// TIA Portal V20 export
ORGANIZATION_BLOCK "Startup"   // OB1030, LAD, Startup
TITLE = "Complete Restart"
// stored: AutoNumber false, IsIECCheckEnabled true, Namespace Unit1.Em5, SetENOAutomatically true
   VAR_INPUT
      LostRetentive : Bool;   // True if retentive data are lost
      LostRTC : Bool;   // True if date and time are lost
   END_VAR
BEGIN

REGION Network 1 (SCL): Build the Absolut Reference Designator
   // Set the Absoult Reference Designator in the Config DB
   IF LEN(IN := "Unit1.Em5.Config".em.referenceDesignator.parent) <> 0 THEN
       "Unit1.Em5.Config".em.referenceDesignator.combined := CONCAT_WSTRING(IN1 := "Unit1.Em5.Config".em.referenceDesignator.parent, IN2 := WSTRING#'.', IN3 := "Unit1.Em5.Config".em.referenceDesignator.relative);
   ELSE
       "Unit1.Em5.Config".em.referenceDesignator.combined := "Unit1.Em5.Config".em.referenceDesignator.relative;
   END_IF;
END_REGION

REGION Network 2 (SCL): Assign axes data
   // This is an example how to assign axes to DB_ANY in DB Config. If you have axes, assign them here. The Config.axis[] variables will be handed over to the control modules. That enables a flexible programming.
   // Assign axes
   "Unit1.Em5.Config".axis[1] := "BA010AZCRDR7_NgManualInputAxisY";
   "Unit1.Em5.Config".axis[2] := "BA010AZCRDR8_MagazineAxisZ";

   // HW_SubModule
   "Unit1.Em5.Config".moduleAccessPoint[1] := "BA010AZCRCU2~BA010AZARCU2_X150~BA010AZCRDR7_ModuleAccessPoint";
   "Unit1.Em5.Config".moduleAccessPoint[2] := "BA010AZCRCU2~BA010AZARCU2_X150~BA010AZCRDR8_ModuleAccessPoint";

   // FB Enable
   "Unit1.Em5.HmiInterface".cmNgAndManualInputAxisY.commands.enableMasterControl := TRUE;
   "Unit1.Em5.HmiInterface".cmMagazineAxisZ.commands.enableMasterControl := TRUE;

   // Assign configuration Homing
   "Unit1.Em5.ControlNodes".cmNgAndManualInputAxisY.commandConfiguration.homing.mode := "Unit1.Em5.HmiInterface".cmNgAndManualInputAxisY.commandConfiguration.homing.mode := 3;
   "Unit1.Em5.ControlNodes".cmMagazineAxisZ.commandConfiguration.homing.mode := "Unit1.Em5.HmiInterface".cmMagazineAxisZ.commandConfiguration.homing.mode := 3;
END_REGION

REGION Network 3 (SCL): CM Config
   // Manual Input Axis Y
   "Unit1.Em5.Config".cmNgAndManualInputAxisY.referenceDesignator := WSTRING#'Manual Input Axis Y';
   "Unit1.Em5.Config".cmNgAndManualInputAxisY.disableAlarms := FALSE;
   "Unit1.Em5.Config".cmNgAndManualInputAxisY.masterControlPopUp := TRUE;


   // Magazine Axis Z
   "Unit1.Em5.Config".cmMagazineAxisZ.referenceDesignator := WSTRING#'Magazine Axis Z';
   "Unit1.Em5.Config".cmMagazineAxisZ.disableAlarms := FALSE;
   "Unit1.Em5.Config".cmMagazineAxisZ.masterControlPopUp := TRUE;


   // Manual Input Cylinder
   "Unit1.Em5.Config".cmNgAndManualInputCylinderUpDown.referenceDesignator := WSTRING#'Manual Input Cylinder';
   "Unit1.Em5.Config".cmNgAndManualInputCylinderUpDown.monitoringLeavingFeedback := T#5s;
   "Unit1.Em5.Config".cmNgAndManualInputCylinderUpDown.monitoringReachingFeedback := T#5s;
   "Unit1.Em5.Config".cmNgAndManualInputCylinderUpDown.monitoringDiscrepancy := T#0ms;
   "Unit1.Em5.Config".cmNgAndManualInputCylinderUpDown.setOutputHomeContinuously := TRUE;
   "Unit1.Em5.Config".cmNgAndManualInputCylinderUpDown.setOutputWorkContinuously := TRUE;
   "Unit1.Em5.Config".cmNgAndManualInputCylinderUpDown.disableHomeCommand := FALSE;
   "Unit1.Em5.Config".cmNgAndManualInputCylinderUpDown.disableFeedbackHomePos := FALSE;
   "Unit1.Em5.Config".cmNgAndManualInputCylinderUpDown.disableFeedbackWorkPos := FALSE;
   "Unit1.Em5.Config".cmNgAndManualInputCylinderUpDown.disableAlarms := FALSE;
   "Unit1.Em5.Config".cmNgAndManualInputCylinderUpDown.resetOutputsOnError := FALSE;
   "Unit1.Em5.Config".cmNgAndManualInputCylinderUpDown.allwaysWaitOnReachingTime := FALSE;


   // Manual Input Vacuum 1
   "Unit1.Em5.Config".cmNgAndManualInputVacuum1OnOff.referenceDesignator := WSTRING#'Manual Input Vacuum1';
   "Unit1.Em5.Config".cmNgAndManualInputVacuum1OnOff.monitoringLeavingFeedback := T#5s;
   "Unit1.Em5.Config".cmNgAndManualInputVacuum1OnOff.monitoringReachingFeedback := T#1s;
   "Unit1.Em5.Config".cmNgAndManualInputVacuum1OnOff.monitoringDiscrepancy := T#0ms;
   "Unit1.Em5.Config".cmNgAndManualInputVacuum1OnOff.setOutputHomeContinuously := FALSE;
   "Unit1.Em5.Config".cmNgAndManualInputVacuum1OnOff.setOutputWorkContinuously := TRUE;
   "Unit1.Em5.Config".cmNgAndManualInputVacuum1OnOff.disableHomeCommand := FALSE;
   "Unit1.Em5.Config".cmNgAndManualInputVacuum1OnOff.disableFeedbackHomePos := TRUE;
   "Unit1.Em5.Config".cmNgAndManualInputVacuum1OnOff.disableFeedbackWorkPos := FALSE;
   "Unit1.Em5.Config".cmNgAndManualInputVacuum1OnOff.disableAlarms := FALSE;
   "Unit1.Em5.Config".cmNgAndManualInputVacuum1OnOff.resetOutputsOnError := FALSE;
   "Unit1.Em5.Config".cmNgAndManualInputVacuum1OnOff.allwaysWaitOnReachingTime := FALSE;


   // Manual Input Vacuum 2
   "Unit1.Em5.Config".cmNgAndManualInputVacuum2OnOff.referenceDesignator := WSTRING#'Manual Input Vacuum2';
   "Unit1.Em5.Config".cmNgAndManualInputVacuum2OnOff.monitoringLeavingFeedback := T#5s;
   "Unit1.Em5.Config".cmNgAndManualInputVacuum2OnOff.monitoringReachingFeedback := T#1s;
   "Unit1.Em5.Config".cmNgAndManualInputVacuum2OnOff.monitoringDiscrepancy := T#0ms;
   "Unit1.Em5.Config".cmNgAndManualInputVacuum2OnOff.setOutputHomeContinuously := FALSE;
   "Unit1.Em5.Config".cmNgAndManualInputVacuum2OnOff.setOutputWorkContinuously := TRUE;
   "Unit1.Em5.Config".cmNgAndManualInputVacuum2OnOff.disableHomeCommand := FALSE;
   "Unit1.Em5.Config".cmNgAndManualInputVacuum2OnOff.disableFeedbackHomePos := TRUE;
   "Unit1.Em5.Config".cmNgAndManualInputVacuum2OnOff.disableFeedbackWorkPos := FALSE;
   "Unit1.Em5.Config".cmNgAndManualInputVacuum2OnOff.disableAlarms := FALSE;
   "Unit1.Em5.Config".cmNgAndManualInputVacuum2OnOff.resetOutputsOnError := FALSE;
   "Unit1.Em5.Config".cmNgAndManualInputVacuum2OnOff.allwaysWaitOnReachingTime := FALSE;


   // Manual Input Vibrator 1
   "Unit1.Em5.Config".cmNgAndManualInputVibrator1OnOff.referenceDesignator := WSTRING#'Manual Input Vibrator1';
   "Unit1.Em5.Config".cmNgAndManualInputVibrator1OnOff.monitoringLeavingFeedback := T#0MS;
   "Unit1.Em5.Config".cmNgAndManualInputVibrator1OnOff.monitoringReachingFeedback := T#1S;
   "Unit1.Em5.Config".cmNgAndManualInputVibrator1OnOff.monitoringDiscrepancy := T#0ms;
   "Unit1.Em5.Config".cmNgAndManualInputVibrator1OnOff.setOutputHomeContinuously := TRUE;
   "Unit1.Em5.Config".cmNgAndManualInputVibrator1OnOff.setOutputWorkContinuously := TRUE;
   "Unit1.Em5.Config".cmNgAndManualInputVibrator1OnOff.disableHomeCommand := FALSE;
   "Unit1.Em5.Config".cmNgAndManualInputVibrator1OnOff.disableFeedbackHomePos := TRUE;
   "Unit1.Em5.Config".cmNgAndManualInputVibrator1OnOff.disableFeedbackWorkPos := TRUE;
   "Unit1.Em5.Config".cmNgAndManualInputVibrator1OnOff.disableAlarms := FALSE;
   "Unit1.Em5.Config".cmNgAndManualInputVibrator1OnOff.resetOutputsOnError := FALSE;
   "Unit1.Em5.Config".cmNgAndManualInputVibrator1OnOff.allwaysWaitOnReachingTime := FALSE;


   // Manual Input Vibrator 2
   "Unit1.Em5.Config".cmNgAndManualInputVibrator2OnOff.referenceDesignator := WSTRING#'Manual Input Vibrator2';
   "Unit1.Em5.Config".cmNgAndManualInputVibrator2OnOff.monitoringLeavingFeedback := T#0MS;
   "Unit1.Em5.Config".cmNgAndManualInputVibrator2OnOff.monitoringReachingFeedback := T#1S;
   "Unit1.Em5.Config".cmNgAndManualInputVibrator2OnOff.monitoringDiscrepancy := T#0ms;
   "Unit1.Em5.Config".cmNgAndManualInputVibrator2OnOff.setOutputHomeContinuously := TRUE;
   "Unit1.Em5.Config".cmNgAndManualInputVibrator2OnOff.setOutputWorkContinuously := TRUE;
   "Unit1.Em5.Config".cmNgAndManualInputVibrator2OnOff.disableHomeCommand := FALSE;
   "Unit1.Em5.Config".cmNgAndManualInputVibrator2OnOff.disableFeedbackHomePos := TRUE;
   "Unit1.Em5.Config".cmNgAndManualInputVibrator2OnOff.disableFeedbackWorkPos := TRUE;
   "Unit1.Em5.Config".cmNgAndManualInputVibrator2OnOff.disableAlarms := FALSE;
   "Unit1.Em5.Config".cmNgAndManualInputVibrator2OnOff.resetOutputsOnError := FALSE;
   "Unit1.Em5.Config".cmNgAndManualInputVibrator2OnOff.allwaysWaitOnReachingTime := FALSE;


   // Magazine Lock Cylinder
   "Unit1.Em5.Config".cmMagazineLockCylinderUpDown.referenceDesignator := WSTRING#'Magazine Lock Cylinder';
   "Unit1.Em5.Config".cmMagazineLockCylinderUpDown.monitoringLeavingFeedback := T#5s;
   "Unit1.Em5.Config".cmMagazineLockCylinderUpDown.monitoringReachingFeedback := T#5s;
   "Unit1.Em5.Config".cmMagazineLockCylinderUpDown.monitoringDiscrepancy := T#0ms;
   "Unit1.Em5.Config".cmMagazineLockCylinderUpDown.setOutputHomeContinuously := TRUE;
   "Unit1.Em5.Config".cmMagazineLockCylinderUpDown.setOutputWorkContinuously := TRUE;
   "Unit1.Em5.Config".cmMagazineLockCylinderUpDown.disableHomeCommand := FALSE;
   "Unit1.Em5.Config".cmMagazineLockCylinderUpDown.disableFeedbackHomePos := FALSE;
   "Unit1.Em5.Config".cmMagazineLockCylinderUpDown.disableFeedbackWorkPos := FALSE;
   "Unit1.Em5.Config".cmMagazineLockCylinderUpDown.disableAlarms := FALSE;
   "Unit1.Em5.Config".cmMagazineLockCylinderUpDown.resetOutputsOnError := FALSE;
   "Unit1.Em5.Config".cmMagazineLockCylinderUpDown.allwaysWaitOnReachingTime := FALSE;


   // Manual Input Magazine Electrode Detection Sensor
   "Unit1.Em5.Config".cmNgAndManaulInputMagazineElectrodeDetectionSensor.referenceDesignator := WSTRING#'DigitalSignal';
   "Unit1.Em5.Config".cmNgAndManaulInputMagazineElectrodeDetectionSensor.onDelay := T#0ms;
   "Unit1.Em5.Config".cmNgAndManaulInputMagazineElectrodeDetectionSensor.offDelay := T#0ms;
   "Unit1.Em5.Config".cmNgAndManaulInputMagazineElectrodeDetectionSensor.default := FALSE;
   "Unit1.Em5.Config".cmNgAndManaulInputMagazineElectrodeDetectionSensor.invertProcessValue := FALSE;
   "Unit1.Em5.Config".cmNgAndManaulInputMagazineElectrodeDetectionSensor.disableAlarms := FALSE;


   // Manual Input Electrode Detection Sensor
   "Unit1.Em5.Config".cmNgAndManualInputElectrodeDetectionSensor.referenceDesignator := WSTRING#'DigitalSignal';
   "Unit1.Em5.Config".cmNgAndManualInputElectrodeDetectionSensor.onDelay := T#0ms;
   "Unit1.Em5.Config".cmNgAndManualInputElectrodeDetectionSensor.offDelay := T#0ms;
   "Unit1.Em5.Config".cmNgAndManualInputElectrodeDetectionSensor.default := FALSE;
   "Unit1.Em5.Config".cmNgAndManualInputElectrodeDetectionSensor.invertProcessValue := FALSE;
   "Unit1.Em5.Config".cmNgAndManualInputElectrodeDetectionSensor.disableAlarms := FALSE;


   // Manual Input Magazine Detection Sensor
   "Unit1.Em5.Config".cmNgAndManualInputMagazineDetectionSensor.referenceDesignator := WSTRING#'DigitalSignal';
   "Unit1.Em5.Config".cmNgAndManualInputMagazineDetectionSensor.onDelay := T#0ms;
   "Unit1.Em5.Config".cmNgAndManualInputMagazineDetectionSensor.offDelay := T#0ms;
   "Unit1.Em5.Config".cmNgAndManualInputMagazineDetectionSensor.default := FALSE;
   "Unit1.Em5.Config".cmNgAndManualInputMagazineDetectionSensor.invertProcessValue := FALSE;
   "Unit1.Em5.Config".cmNgAndManualInputMagazineDetectionSensor.disableAlarms := FALSE;


   // Manual Input Magazine Full Sensor
   "Unit1.Em5.Config".cmNgAndManualInputMagazineFullSensor.referenceDesignator := WSTRING#'DigitalSignal';
   "Unit1.Em5.Config".cmNgAndManualInputMagazineFullSensor.onDelay := T#0ms;
   "Unit1.Em5.Config".cmNgAndManualInputMagazineFullSensor.offDelay := T#0ms;
   "Unit1.Em5.Config".cmNgAndManualInputMagazineFullSensor.default := FALSE;
   "Unit1.Em5.Config".cmNgAndManualInputMagazineFullSensor.invertProcessValue := FALSE;
   "Unit1.Em5.Config".cmNgAndManualInputMagazineFullSensor.disableAlarms := FALSE;


   // Softcam
   //HmiInterface.cm.softcam.ngAndManualInput.UnitName := WSTRING#'mm';
   //HmiInterface.cm.softcam.magazine.UnitName := WSTRING#'mm';
END_REGION
END_ORGANIZATION_BLOCK
